// SIMATIC S7-200 project (STEP 7-Micro/WIN), CPU 226 CN REL 02.01

SYMBOL_TABLE 设备点名
烟气温度报警延时         T200
烟气温度报警限值         VD648
烟气压力保持数值         VD640
烟气流量保持数值         VD644
烟气温度保持数值         VD636
测量持续时间           T42
中间点3             V5010.2
中间点2             V5010.1
定时反吹持续时间         T39
后吹扫持续时间          T41
中间点1             V5010.0
干基折算粉尘浓度         VD632
测量               V1015.7
工况下烟气流量          VD608
烟气流速             VD616
Analyzer_Cali_FTE V6000.5
定时反吹_FTE         V6000.4
测量_FTE           V6000.3
后吹扫_FTE          V6000.2
采集背景_FTE         V6000.1
前吹扫_FTE          V6000.0
当前动作字符串输出        VB6100
Analyzer_Cali_STATU V1016.3
烟气温度低报警_STATU    V1012.6
维护切换_M           M1.0
手动_自动_M          M1.1
系统待机_M           M1.2
停止蜂鸣器_M          M1.3
手动启动             M1.4
探头反吹_M           M2.0
探头通零气_M          M2.1
探头通标气_M          M2.2
分析仪反吹_M          M2.3
分析仪通零气_M         M2.4
分析仪通标气_M         M2.5
手动采集背景_M         M2.6
测量_M             M2.7
蜂鸣器停止间隔时间        T40
报警指示灯_img        V1000.0
维护指示灯_img        V1000.1
运行指示灯_img        V1000.2
蜂鸣器_img          V1000.3
DCS报警信号_img      V1000.4
DCS运行信号_img      V1000.5
DCS维护信号_img      V1000.6
DCS待机信号_img      V1000.7
HOFI反吹电磁阀_img    V1001.0
三通电磁阀_img        V1001.1
氮气电磁阀_img        V1001.2
标气电磁阀_img        V1001.3
常开两通电磁阀_img      V1001.4
报警消除信号_img       V1004.0
DCS控制待机信号        V1004.2
探头反吹_ACT         V1006.0
探头通零气_ACT        V1006.1
探头通标气_ACT        V1006.2
分析仪反吹_ACT        V1006.3
分析仪通零气_ACT       V1006.4
分析仪通标气_ACT       V1006.5
采集背景_ACT         V1006.6
分析仪测量_ACT        V1006.7
探头后吹扫_ACT        V1007.0
分析仪前吹扫_ACT       V1007.1
定时反吹_ACT         V1007.2
Analyzer_Calibartion V1007.3
手动_自动_ACT        V1008.0
停止蜂鸣器_ACT        V1008.1
维护切换_ACT         V1008.4
待机_运行_ACT        V1008.5
启动报警_ACT         V1008.6
系统待机_ACT         V1008.7
系统运行_STATU       V1009.3
系统维护_STATU       V1009.4
系统报警_STATU       V1009.5
系统待机_STATU       V1009.6
手动_自动_STATU      V1010.6
蜂鸣器停止_运行_STATU   V1010.7
HOFI压力报警_STATU   V1011.0
HOFI温度报警_STATU   V1011.1
MDS压力报警_STATU    V1011.2
N2压力报警_STATU     V1011.3
粉尘仪报警_STATU      V1011.4
气路模块温度报警_STATU   V1011.5
加热管线温度报警_STATU   V1011.6
检测室温度报警_STATU    V1011.7
Reference失败报警_STATU V1012.0
检测室压力报警_STATU    V1012.1
文丘里压力报警_STATU    V1012.2
分析仪参数报警_STATU    V1012.3
分析仪报警_STATU      V1012.4
采样系统报警_STATU     V1012.5
联机通讯状警_STATU     V1012.7
采集背景_STATU       V1015.6
后吹扫_STATU        V1016.0
前吹扫_STATU        V1016.1
定时反吹_STATU       V1016.2
蜂鸣器启动中间变量        V5002.0
HCL折算            VD524
SO2折算            VD528
NOx折算            VD532
NH3折算            VD536
NO折算             VD540
NO2折算            VD544
SO2实测值           VD548
HF折算             VD552
CO折算             VD556
CO2折算            VD560
NOX实测值           VD564
水分含量             VD568
湿氧浓度             VD576
检测室压力            VD580
文丘里压力            VD584
烟气温度             VD592
烟气压力             VD596
烟气压差             VD600
粉尘浓度             VD604
干基标准烟气流量         VD620
标态粉尘浓度           VD624
干氧浓度             VD628
检测室压力_img        VW900
文丘里压力_img        VW902
湿氧浓度_img         VW904
烟气温度_img         VW906
烟气压差_img         VW908
烟气压力_img         VW910
粉尘浓度_img         VW912
END_SYMBOL_TABLE

ORGANIZATION_BLOCK Main:OB1
TITLE=
// //增加氧气修正及烟气流量，粉尘修正的计算
// //模拟量输出量程设置
// //增加定时反吹定时时间 配合组态用于MBGAS3000驱动
// //Define Action子程序，增加报警状态点 V1009.5  网络16,17
// //Define Action子程序，修改1008.5为待机_运行控制点，输出状态为系统待机， 网络14,15
// //Operation & Remove Operation子程序增加V1000.7信号的置位与复位
// 
// //修改干基计算子模块为标态计算
// 
// //采样系统报警时也可执行待机动作
// 
// //增加profibusDP数据通信功能
// 
// 
BEGIN
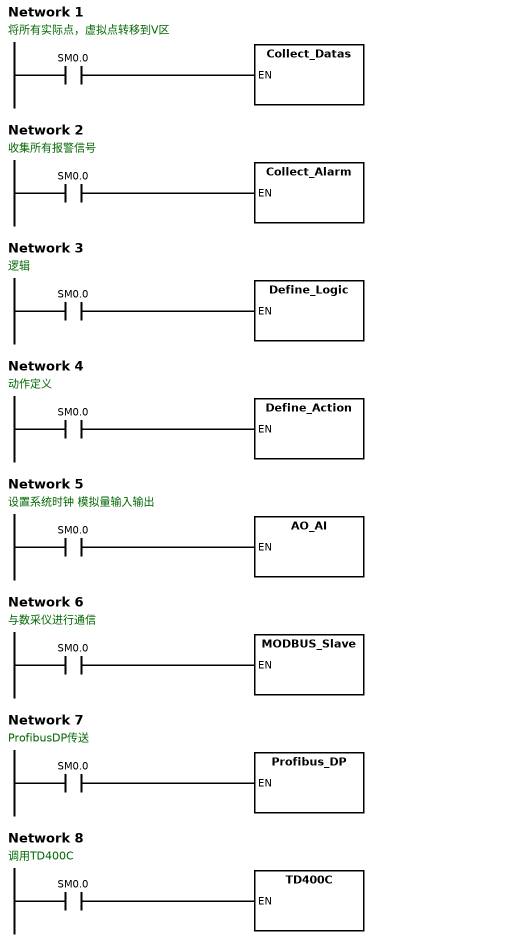
Network 1
// 将所有实际点，虚拟点转移到V区
LD     SM0.0
CALL   Collect_Datas:SBR7
Network 2
// 收集所有报警信号
LD     SM0.0
CALL   Collect_Alarm:SBR8
Network 3
// 逻辑
LD     SM0.0
CALL   Define_Logic:SBR10
Network 4
// 动作定义
LD     SM0.0
CALL   Define_Action:SBR9
Network 5
// 设置系统时钟 模拟量输入输出
LD     SM0.0
CALL   AO_AI:SBR15
Network 6
// 与数采仪进行通信
LD     SM0.0
CALL   MODBUS_Slave:SBR21
Network 7
// ProfibusDP传送
LD     SM0.0
CALL   Profibus_DP:SBR25
Network 8
// 调用TD400C
LD     SM0.0
CALL   TD400C:SBR16
END_ORGANIZATION_BLOCK

// SBR0: protected block, not included

SUBROUTINE_BLOCK Alarm:SBR1
TITLE=报警执行动作
BEGIN
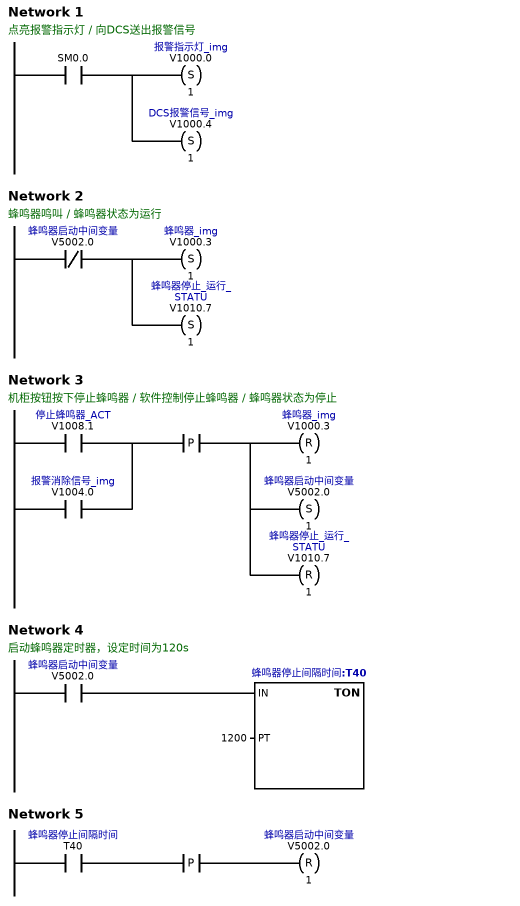
Network 1
// 点亮报警指示灯
// 向DCS送出报警信号
LD     SM0.0
S      报警指示灯_img:V1000.0, 1
S      DCS报警信号_img:V1000.4, 1
Network 2
// 蜂鸣器鸣叫
// 蜂鸣器状态为运行
LDN    蜂鸣器启动中间变量:V5002.0
S      蜂鸣器_img:V1000.3, 1
S      蜂鸣器停止_运行_STATU:V1010.7, 1
Network 3
// 机柜按钮按下停止蜂鸣器
// 软件控制停止蜂鸣器
// 蜂鸣器状态为停止
LD     停止蜂鸣器_ACT:V1008.1
O      报警消除信号_img:V1004.0
EU
R      蜂鸣器_img:V1000.3, 1
S      蜂鸣器启动中间变量:V5002.0, 1
R      蜂鸣器停止_运行_STATU:V1010.7, 1
Network 4
// 启动蜂鸣器定时器，设定时间为120s
LD     蜂鸣器启动中间变量:V5002.0
TON    蜂鸣器停止间隔时间:T40, 1200
Network 5
LD     蜂鸣器停止间隔时间:T40
EU
R      蜂鸣器启动中间变量:V5002.0, 1
END_SUBROUTINE_BLOCK

SUBROUTINE_BLOCK Remove_Alarm:SBR2
TITLE=报警消除后执行动作
BEGIN
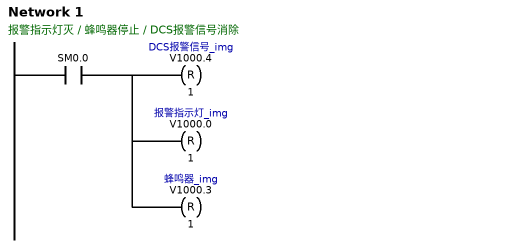
Network 1
// 报警指示灯灭
// 蜂鸣器停止
// DCS报警信号消除
LD     SM0.0
R      DCS报警信号_img:V1000.4, 1
R      报警指示灯_img:V1000.0, 1
R      蜂鸣器_img:V1000.3, 1
END_SUBROUTINE_BLOCK

SUBROUTINE_BLOCK Operation:SBR3
TITLE=子程序注释
BEGIN
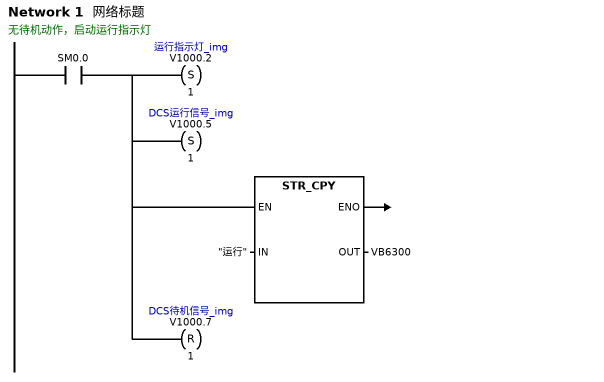
Network 1 // 网络标题
// 无待机动作，启动运行指示灯
LD     SM0.0
S      运行指示灯_img:V1000.2, 1
S      DCS运行信号_img:V1000.5, 1
SCPY   "运行", VB6300
R      DCS待机信号_img:V1000.7, 1
END_SUBROUTINE_BLOCK

SUBROUTINE_BLOCK Remove_Operation:SBR4
TITLE=子程序注释
BEGIN
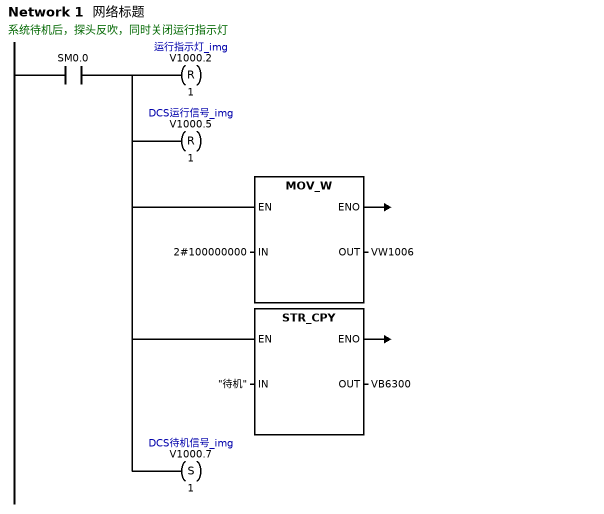
Network 1 // 网络标题
// 系统待机后，探头反吹，同时关闭运行指示灯
LD     SM0.0
R      运行指示灯_img:V1000.2, 1
R      DCS运行信号_img:V1000.5, 1
MOVW   2#100000000, VW1006
SCPY   "待机", VB6300
S      DCS待机信号_img:V1000.7, 1
Network 11 // 网络标题
// 网络注释
END_SUBROUTINE_BLOCK

SUBROUTINE_BLOCK Maintenance:SBR5
TITLE=子程序注释
BEGIN
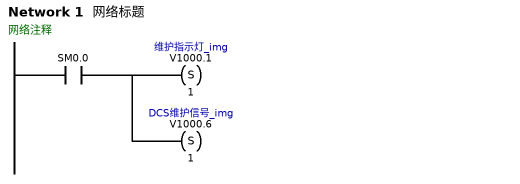
Network 1 // 网络标题
// 网络注释
LD     SM0.0
S      维护指示灯_img:V1000.1, 1
S      DCS维护信号_img:V1000.6, 1
END_SUBROUTINE_BLOCK

SUBROUTINE_BLOCK Remove_Maintenance:SBR6
TITLE=子程序注释
BEGIN
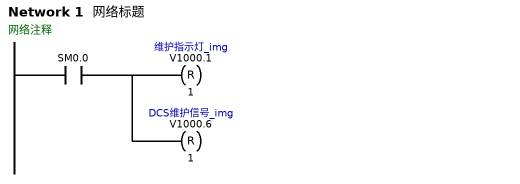
Network 1 // 网络标题
// 网络注释
LD     SM0.0
R      维护指示灯_img:V1000.1, 1
R      DCS维护信号_img:V1000.6, 1
END_SUBROUTINE_BLOCK

SUBROUTINE_BLOCK Collect_Datas:SBR7
TITLE=数据转移V区
BEGIN
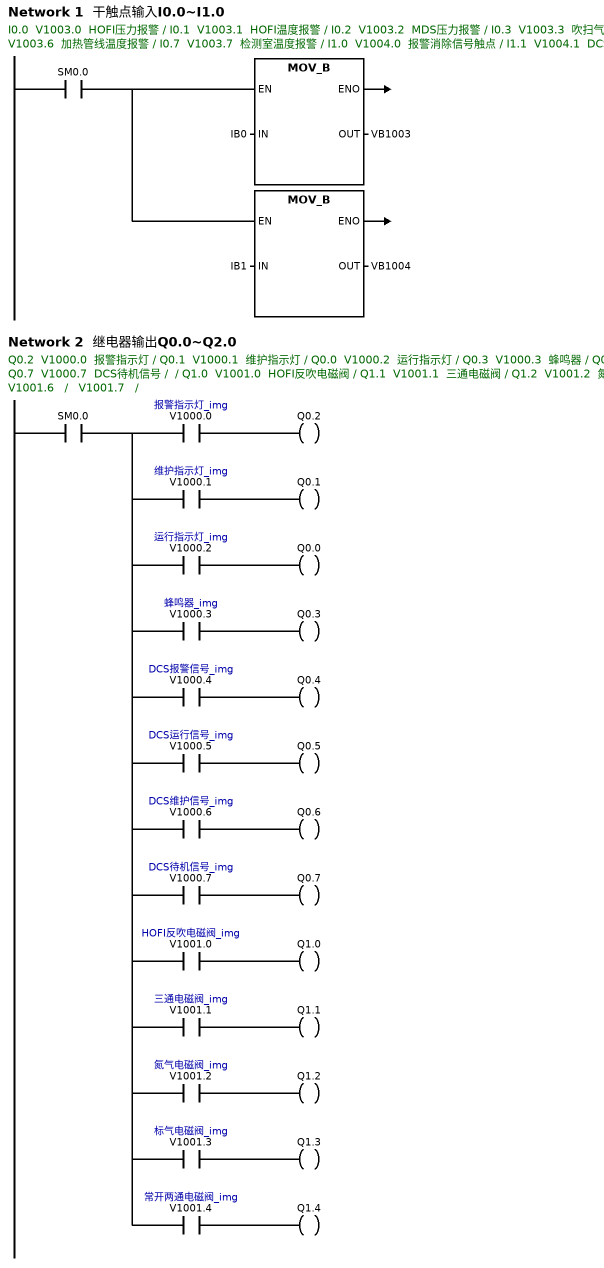
Network 1 // 干触点输入I0.0~I1.0
// I0.0	V1003.0	HOFI压力报警
// I0.1	V1003.1	HOFI温度报警
// I0.2	V1003.2	MDS压力报警
// I0.3	V1003.3	吹扫气体发生器输出压力报警
// I0.4	V1003.4	粉尘仪报警
// I0.5	V1003.5	分析仪采样模块温度报警
// I0.6	V1003.6	加热管线温度报警
// I0.7	V1003.7	检测室温度报警
// I1.0	V1004.0	报警消除信号触点
// I1.1	V1004.1	DCS控制系统采样信号
// I1.2	V1004.2	DCS控制系统待机信号
LD     SM0.0
MOVB   IB0, VB1003
MOVB   IB1, VB1004
Network 2 // 继电器输出Q0.0~Q2.0
// Q0.2	V1000.0	报警指示灯
// Q0.1	V1000.1	维护指示灯
// Q0.0	V1000.2	运行指示灯
// Q0.3	V1000.3	蜂鸣器
// Q0.4	V1000.4	DCS报警信号
// Q0.5	V1000.5	DCS运行信号
// Q0.6	V1000.6	DCS维护信号
// Q0.7	V1000.7	DCS待机信号
// 
// Q1.0	V1001.0	HOFI反吹电磁阀
// Q1.1	V1001.1	三通电磁阀
// Q1.2	V1001.2	氮气电磁阀
// Q1.3	V1001.3	标气电磁阀
// Q1.4	V1001.4	常开两通电磁阀
// 	V1001.5	
// 	V1001.6	
// 	V1001.7	
// 
LD     SM0.0
LPS
A      报警指示灯_img:V1000.0
=      Q0.2
LRD
A      维护指示灯_img:V1000.1
=      Q0.1
LRD
A      运行指示灯_img:V1000.2
=      Q0.0
LRD
A      蜂鸣器_img:V1000.3
=      Q0.3
LRD
A      DCS报警信号_img:V1000.4
=      Q0.4
LRD
A      DCS运行信号_img:V1000.5
=      Q0.5
LRD
A      DCS维护信号_img:V1000.6
=      Q0.6
LRD
A      DCS待机信号_img:V1000.7
=      Q0.7
LRD
A      HOFI反吹电磁阀_img:V1001.0
=      Q1.0
LRD
A      三通电磁阀_img:V1001.1
=      Q1.1
LRD
A      氮气电磁阀_img:V1001.2
=      Q1.2
LRD
A      标气电磁阀_img:V1001.3
=      Q1.3
LPP
A      常开两通电磁阀_img:V1001.4
=      Q1.4
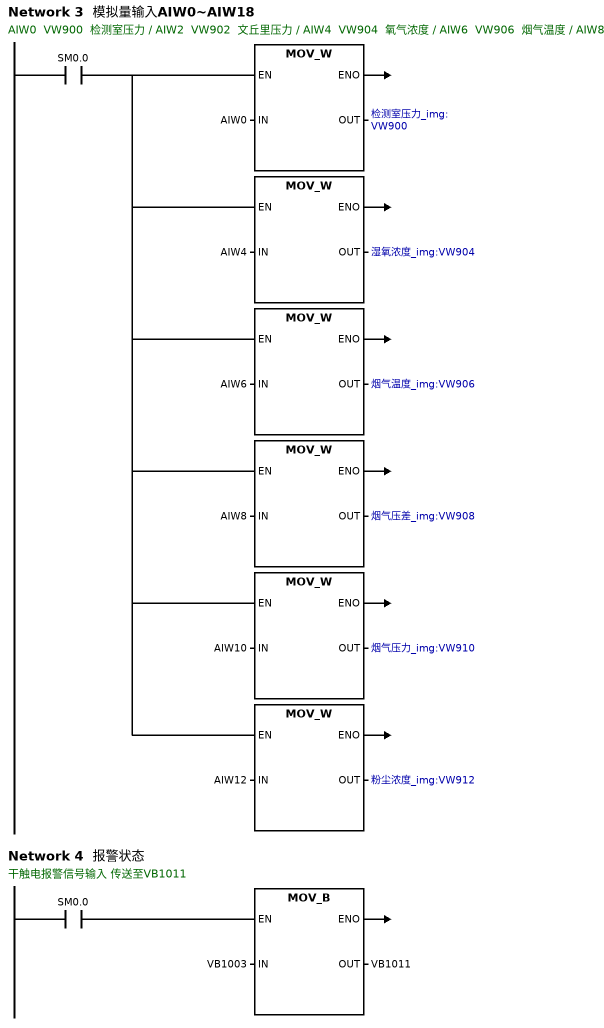
Network 3 // 模拟量输入AIW0~AIW18
// AIW0	VW900	检测室压力
// AIW2	VW902	文丘里压力
// AIW4	VW904	氧气浓度
// AIW6	VW906	烟气温度
// AIW8	VW908	烟气压差
// AIW10	VW910	烟气压力
// AIW12	VW912	粉尘浓度/不透光度
// 
LD     SM0.0
MOVW   AIW0, 检测室压力_img:VW900
MOVW   AIW4, 湿氧浓度_img:VW904
MOVW   AIW6, 烟气温度_img:VW906
MOVW   AIW8, 烟气压差_img:VW908
MOVW   AIW10, 烟气压力_img:VW910
MOVW   AIW12, 粉尘浓度_img:VW912
Network 4 // 报警状态
// 干触电报警信号输入 传送至VB1011
LD     SM0.0
MOVB   VB1003, VB1011
END_SUBROUTINE_BLOCK

SUBROUTINE_BLOCK Collect_Alarm:SBR8
TITLE=
BEGIN
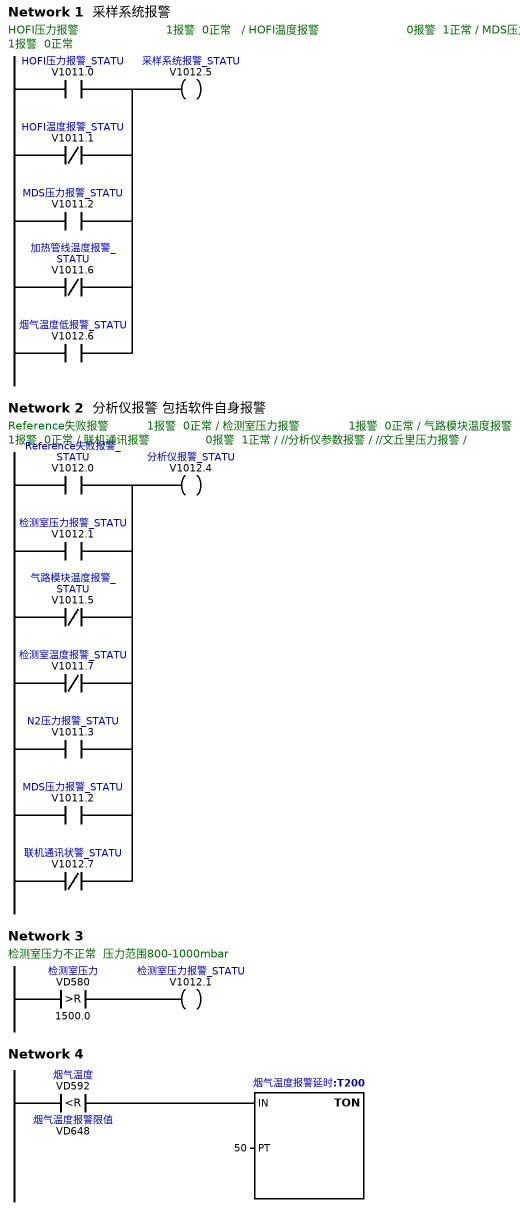
Network 1 // 采样系统报警
// HOFI压力报警                         1报警  0正常  
// HOFI温度报警                         0报警  1正常
// MDS压力报警                          1报警  0正常
// 加热管线温度报警                     0报警  1正常
// 烟气温度低                           1报警  0正常
LD     HOFI压力报警_STATU:V1011.0
ON     HOFI温度报警_STATU:V1011.1
O      MDS压力报警_STATU:V1011.2
ON     加热管线温度报警_STATU:V1011.6
O      烟气温度低报警_STATU:V1012.6
=      采样系统报警_STATU:V1012.5
Network 2 // 分析仪报警 包括软件自身报警
// Reference失败报警           1报警  0正常
// 检测室压力报警              1报警  0正常
// 气路模块温度报警            0报警  1正常
// 检测室温度报警              0报警  1正常
// N2压力报警                  1报警  0正常
// MDS压力报警                 1报警  0正常
// 联机通讯报警                0报警  1正常
// //分析仪参数报警
// //文丘里压力报警
// 
LD     Reference失败报警_STATU:V1012.0
O      检测室压力报警_STATU:V1012.1
ON     气路模块温度报警_STATU:V1011.5
ON     检测室温度报警_STATU:V1011.7
O      N2压力报警_STATU:V1011.3
O      MDS压力报警_STATU:V1011.2
ON     联机通讯状警_STATU:V1012.7
=      分析仪报警_STATU:V1012.4
Network 3
// 检测室压力不正常  压力范围800-1000mbar
LDR>   检测室压力:VD580, 1500.0
=      检测室压力报警_STATU:V1012.1
Network 4
LDR<   烟气温度:VD592, 烟气温度报警限值:VD648
TON    烟气温度报警延时:T200, 50
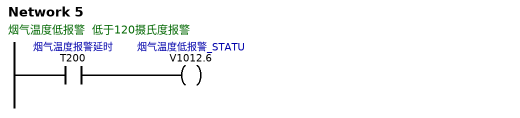
Network 5
// 烟气温度低报警  低于120摄氏度报警
LD     烟气温度报警延时:T200
=      烟气温度低报警_STATU:V1012.6
END_SUBROUTINE_BLOCK

SUBROUTINE_BLOCK Define_Action:SBR9
TITLE=
BEGIN
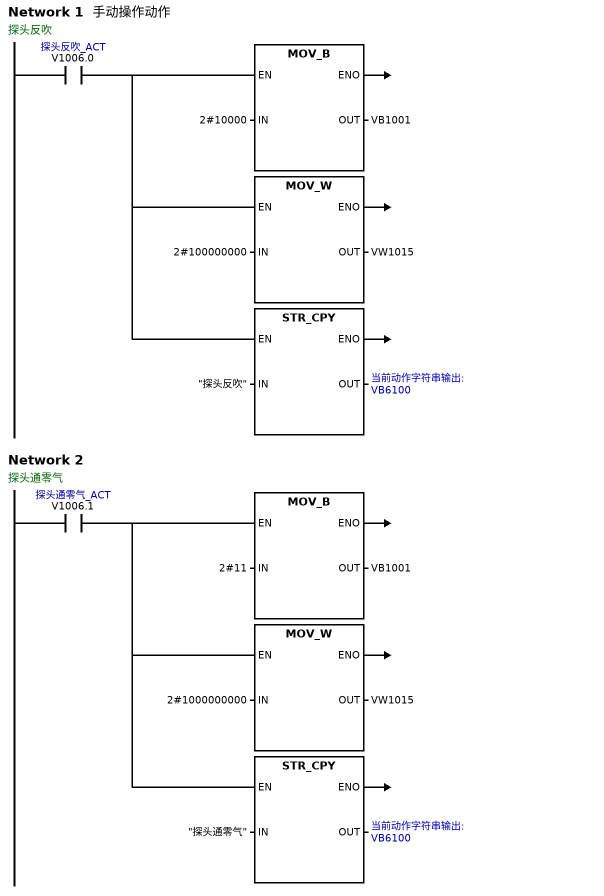
Network 1 // 手动操作动作
// 探头反吹
LD     探头反吹_ACT:V1006.0
MOVB   2#10000, VB1001
MOVW   2#100000000, VW1015
SCPY   "探头反吹", 当前动作字符串输出:VB6100
Network 2
// 探头通零气
LD     探头通零气_ACT:V1006.1
MOVB   2#11, VB1001
MOVW   2#1000000000, VW1015
SCPY   "探头通零气", 当前动作字符串输出:VB6100
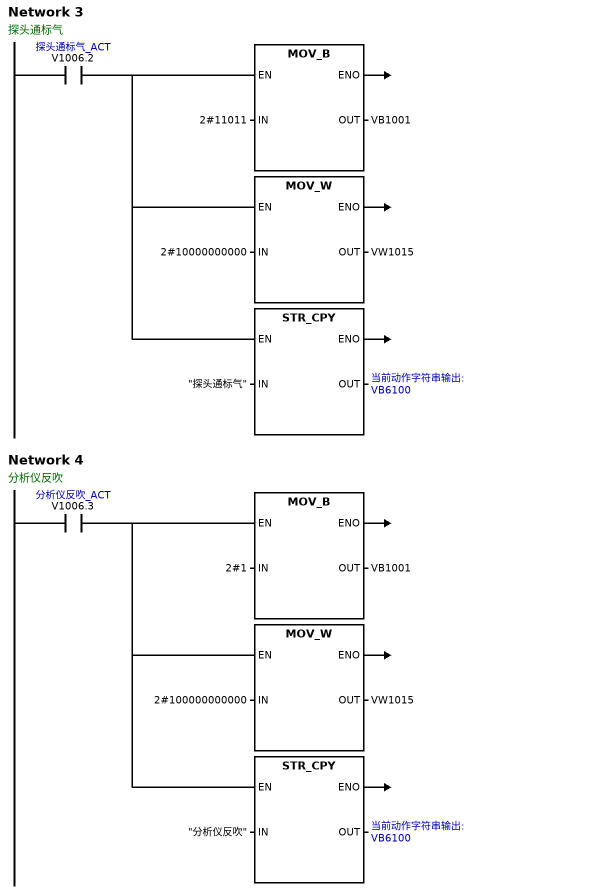
Network 3
// 探头通标气
LD     探头通标气_ACT:V1006.2
MOVB   2#11011, VB1001
MOVW   2#10000000000, VW1015
SCPY   "探头通标气", 当前动作字符串输出:VB6100
Network 4
// 分析仪反吹
LD     分析仪反吹_ACT:V1006.3
MOVB   2#1, VB1001
MOVW   2#100000000000, VW1015
SCPY   "分析仪反吹", 当前动作字符串输出:VB6100
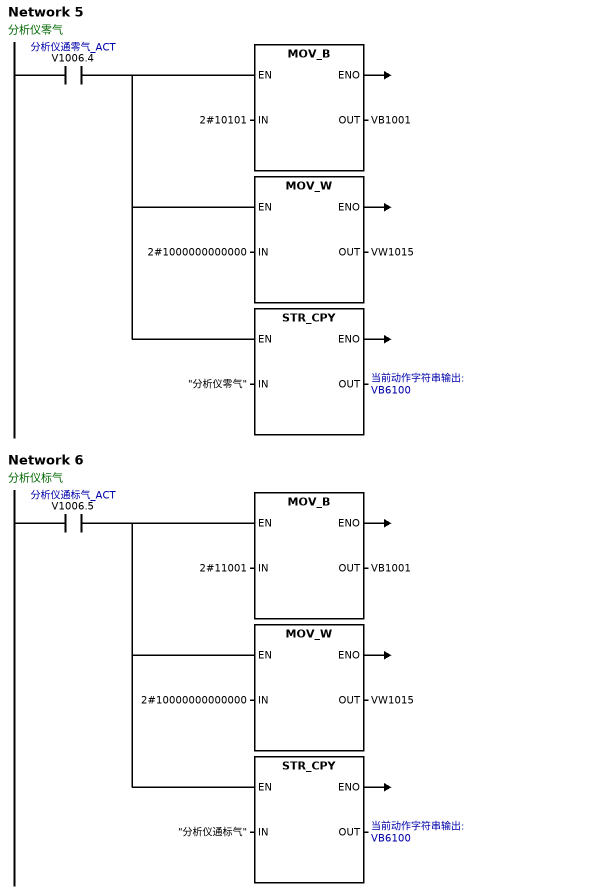
Network 5
// 分析仪零气
LD     分析仪通零气_ACT:V1006.4
MOVB   2#10101, VB1001
MOVW   2#1000000000000, VW1015
SCPY   "分析仪零气", 当前动作字符串输出:VB6100
Network 6
// 分析仪标气
LD     分析仪通标气_ACT:V1006.5
MOVB   2#11001, VB1001
MOVW   2#10000000000000, VW1015
SCPY   "分析仪通标气", 当前动作字符串输出:VB6100
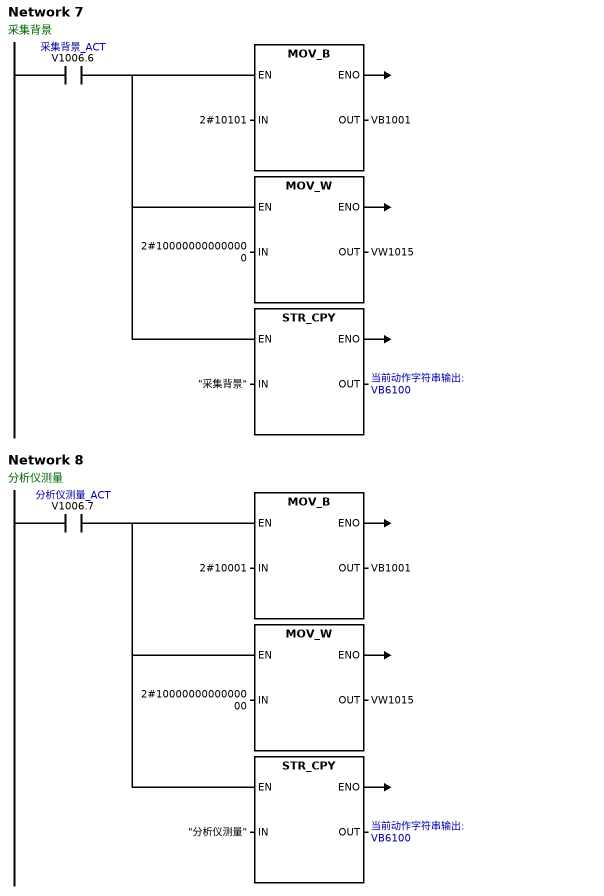
Network 7
// 采集背景
LD     采集背景_ACT:V1006.6
MOVB   2#10101, VB1001
MOVW   2#100000000000000, VW1015
SCPY   "采集背景", 当前动作字符串输出:VB6100
Network 8
// 分析仪测量
LD     分析仪测量_ACT:V1006.7
MOVB   2#10001, VB1001
MOVW   2#1000000000000000, VW1015
SCPY   "分析仪测量", 当前动作字符串输出:VB6100
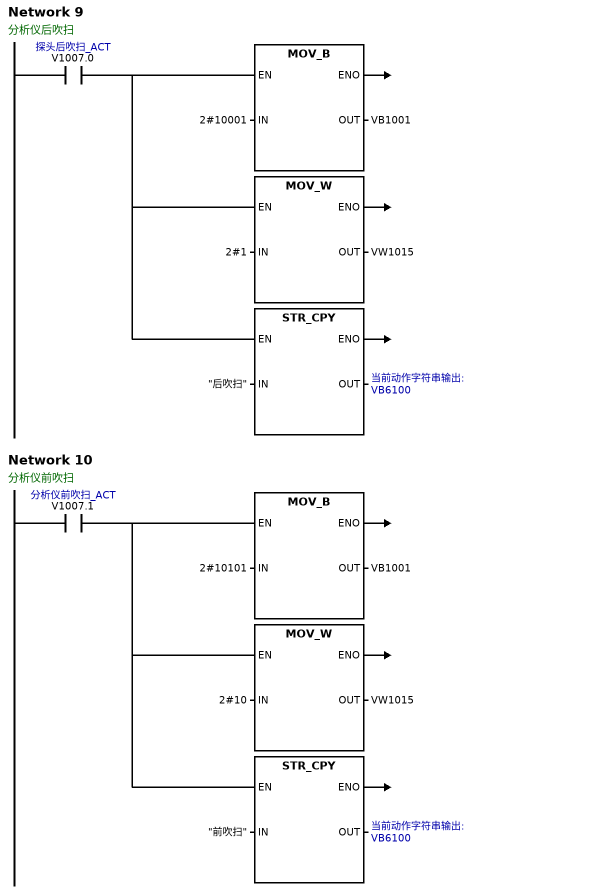
Network 9
// 分析仪后吹扫
LD     探头后吹扫_ACT:V1007.0
MOVB   2#10001, VB1001
MOVW   2#1, VW1015
SCPY   "后吹扫", 当前动作字符串输出:VB6100
Network 10
// 分析仪前吹扫
LD     分析仪前吹扫_ACT:V1007.1
MOVB   2#10101, VB1001
MOVW   2#10, VW1015
SCPY   "前吹扫", 当前动作字符串输出:VB6100
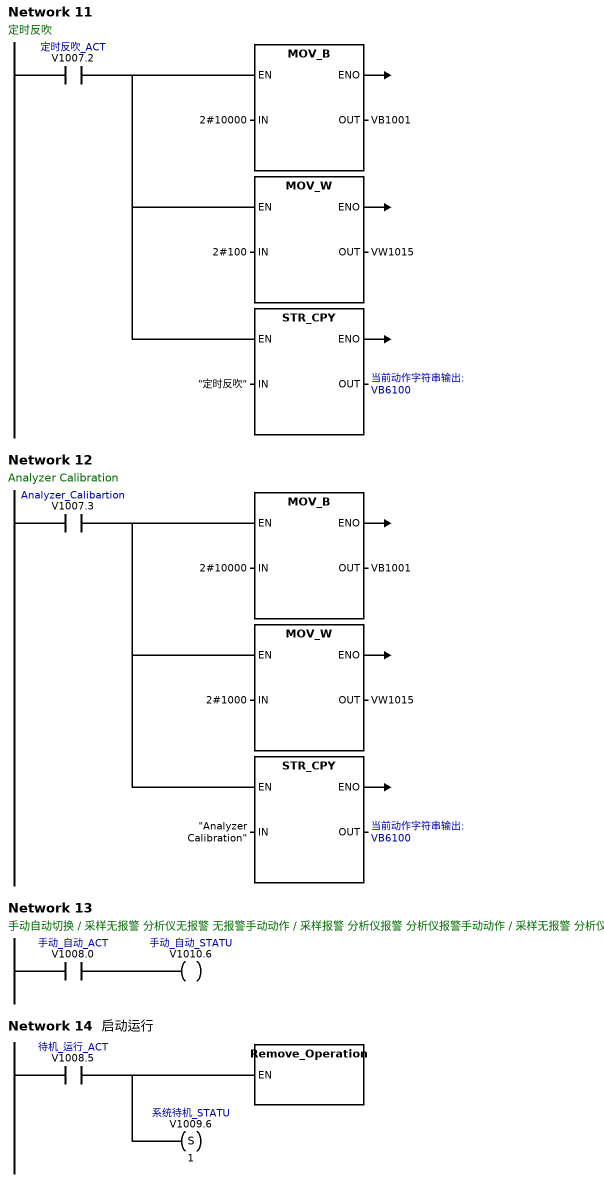
Network 11
// 定时反吹
LD     定时反吹_ACT:V1007.2
MOVB   2#10000, VB1001
MOVW   2#100, VW1015
SCPY   "定时反吹", 当前动作字符串输出:VB6100
Network 12
// Analyzer Calibration
LD     Analyzer_Calibartion:V1007.3
MOVB   2#10000, VB1001
MOVW   2#1000, VW1015
SCPY   "Analyzer Calibration", 当前动作字符串输出:VB6100
Network 13
// 手动自动切换
// 采样无报警 分析仪无报警 无报警手动动作
// 采样报警 分析仪报警 分析仪报警手动动作
// 采样无报警 分析仪报警 分析仪报警手动动作
// 采样报警 分析仪无报警 探头报警手动动作
LD     手动_自动_ACT:V1008.0
=      手动_自动_STATU:V1010.6
Network 14 // 启动运行
LD     待机_运行_ACT:V1008.5
CALL   Remove_Operation:SBR4
S      系统待机_STATU:V1009.6, 1
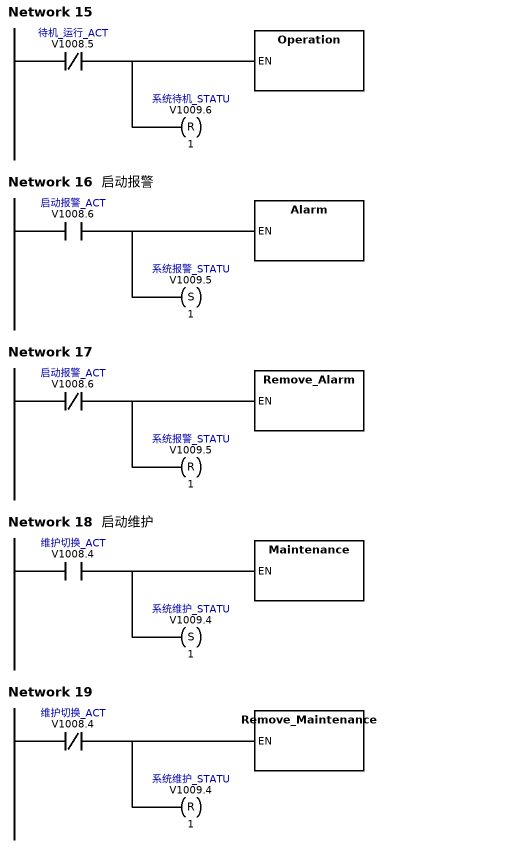
Network 15
LDN    待机_运行_ACT:V1008.5
CALL   Operation:SBR3
R      系统待机_STATU:V1009.6, 1
Network 16 // 启动报警
LD     启动报警_ACT:V1008.6
CALL   Alarm:SBR1
S      系统报警_STATU:V1009.5, 1
Network 17
LDN    启动报警_ACT:V1008.6
CALL   Remove_Alarm:SBR2
R      系统报警_STATU:V1009.5, 1
Network 18 // 启动维护
LD     维护切换_ACT:V1008.4
CALL   Maintenance:SBR5
S      系统维护_STATU:V1009.4, 1
Network 19
LDN    维护切换_ACT:V1008.4
CALL   Remove_Maintenance:SBR6
R      系统维护_STATU:V1009.4, 1
END_SUBROUTINE_BLOCK

SUBROUTINE_BLOCK Define_Logic:SBR10
TITLE=
BEGIN
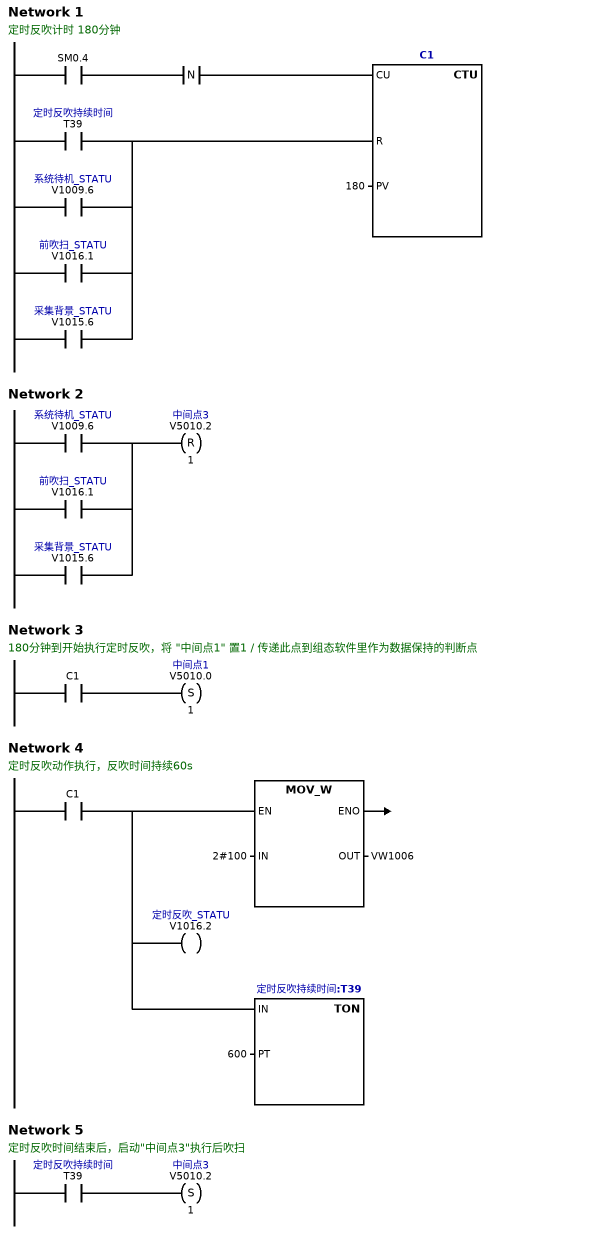
Network 1
// 定时反吹计时 180分钟
LD     SM0.4
ED
LD     定时反吹持续时间:T39
O      系统待机_STATU:V1009.6
O      前吹扫_STATU:V1016.1
O      采集背景_STATU:V1015.6
CTU    C1, 180
Network 2
LD     系统待机_STATU:V1009.6
O      前吹扫_STATU:V1016.1
O      采集背景_STATU:V1015.6
R      中间点3:V5010.2, 1
Network 3
// 180分钟到开始执行定时反吹，将 "中间点1" 置1
// 传递此点到组态软件里作为数据保持的判断点
LD     C1
S      中间点1:V5010.0, 1
Network 4
// 定时反吹动作执行，反吹时间持续60s
LD     C1
MOVW   2#100, VW1006
=      定时反吹_STATU:V1016.2
TON    定时反吹持续时间:T39, 600
Network 5
// 定时反吹时间结束后，启动"中间点3"执行后吹扫
LD     定时反吹持续时间:T39
S      中间点3:V5010.2, 1
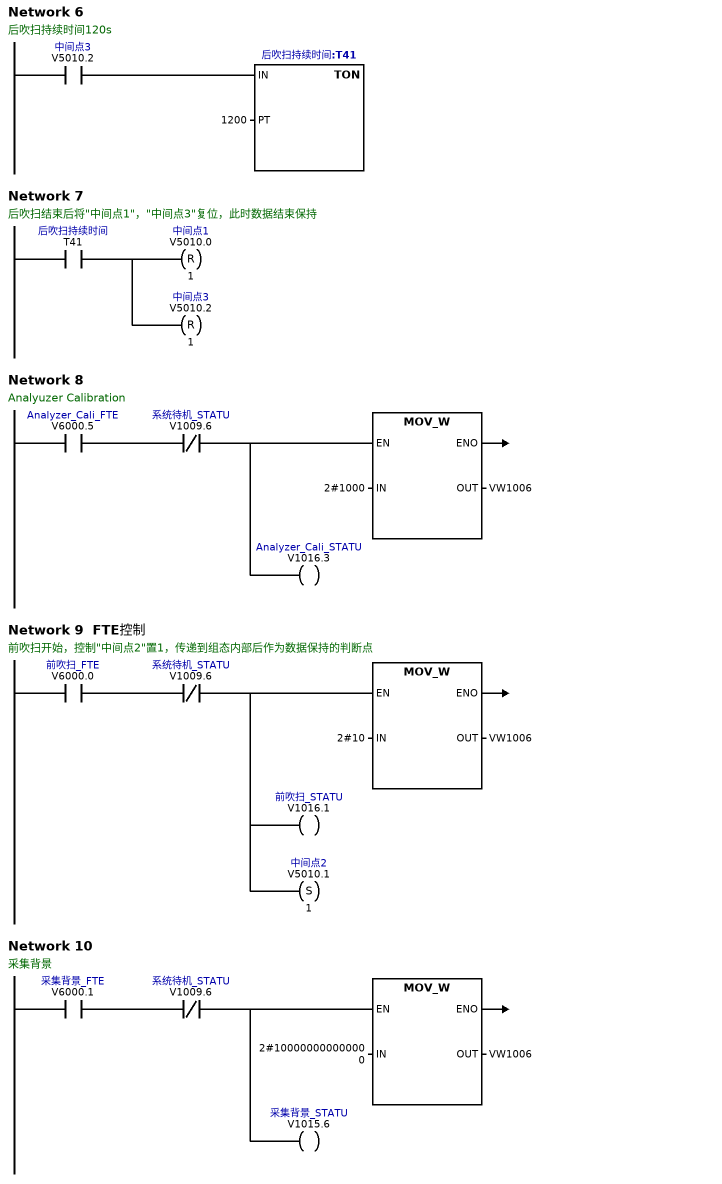
Network 6
// 后吹扫持续时间120s
LD     中间点3:V5010.2
TON    后吹扫持续时间:T41, 1200
Network 7
// 后吹扫结束后将"中间点1"，"中间点3"复位，此时数据结束保持
LD     后吹扫持续时间:T41
R      中间点1:V5010.0, 1
R      中间点3:V5010.2, 1
Network 8
// Analyuzer Calibration
LD     Analyzer_Cali_FTE:V6000.5
AN     系统待机_STATU:V1009.6
MOVW   2#1000, VW1006
=      Analyzer_Cali_STATU:V1016.3
Network 9 // FTE控制
// 前吹扫开始，控制"中间点2"置1，传递到组态内部后作为数据保持的判断点
LD     前吹扫_FTE:V6000.0
AN     系统待机_STATU:V1009.6
MOVW   2#10, VW1006
=      前吹扫_STATU:V1016.1
S      中间点2:V5010.1, 1
Network 10
// 采集背景
LD     采集背景_FTE:V6000.1
AN     系统待机_STATU:V1009.6
MOVW   2#100000000000000, VW1006
=      采集背景_STATU:V1015.6
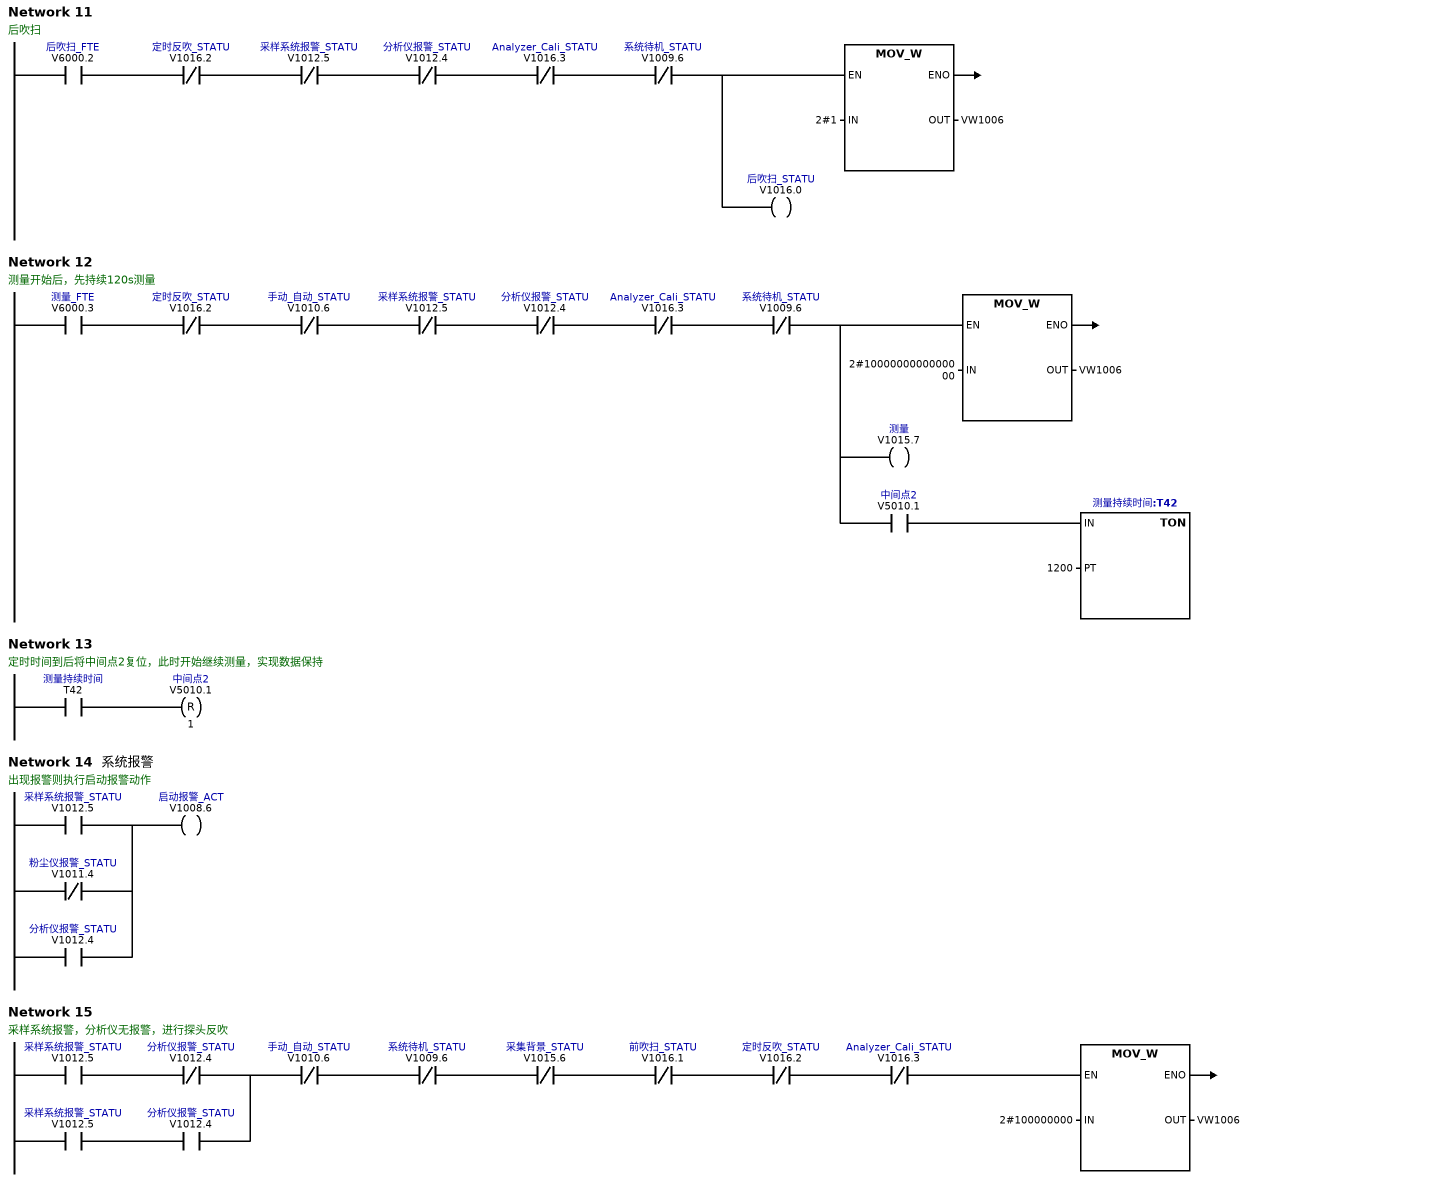
Network 11
// 后吹扫
LD     后吹扫_FTE:V6000.2
AN     定时反吹_STATU:V1016.2
AN     采样系统报警_STATU:V1012.5
AN     分析仪报警_STATU:V1012.4
AN     Analyzer_Cali_STATU:V1016.3
AN     系统待机_STATU:V1009.6
MOVW   2#1, VW1006
=      后吹扫_STATU:V1016.0
Network 12
// 测量开始后，先持续120s测量
LD     测量_FTE:V6000.3
AN     定时反吹_STATU:V1016.2
AN     手动_自动_STATU:V1010.6
AN     采样系统报警_STATU:V1012.5
AN     分析仪报警_STATU:V1012.4
AN     Analyzer_Cali_STATU:V1016.3
AN     系统待机_STATU:V1009.6
MOVW   2#1000000000000000, VW1006
=      测量:V1015.7
A      中间点2:V5010.1
TON    测量持续时间:T42, 1200
Network 13
// 定时时间到后将中间点2复位，此时开始继续测量，实现数据保持
LD     测量持续时间:T42
R      中间点2:V5010.1, 1
Network 14 // 系统报警
// 出现报警则执行启动报警动作
LD     采样系统报警_STATU:V1012.5
ON     粉尘仪报警_STATU:V1011.4
O      分析仪报警_STATU:V1012.4
=      启动报警_ACT:V1008.6
Network 15
// 采样系统报警，分析仪无报警，进行探头反吹
LD     采样系统报警_STATU:V1012.5
AN     分析仪报警_STATU:V1012.4
LD     采样系统报警_STATU:V1012.5
A      分析仪报警_STATU:V1012.4
OLD
AN     手动_自动_STATU:V1010.6
AN     系统待机_STATU:V1009.6
AN     采集背景_STATU:V1015.6
AN     前吹扫_STATU:V1016.1
AN     定时反吹_STATU:V1016.2
AN     Analyzer_Cali_STATU:V1016.3
MOVW   2#100000000, VW1006
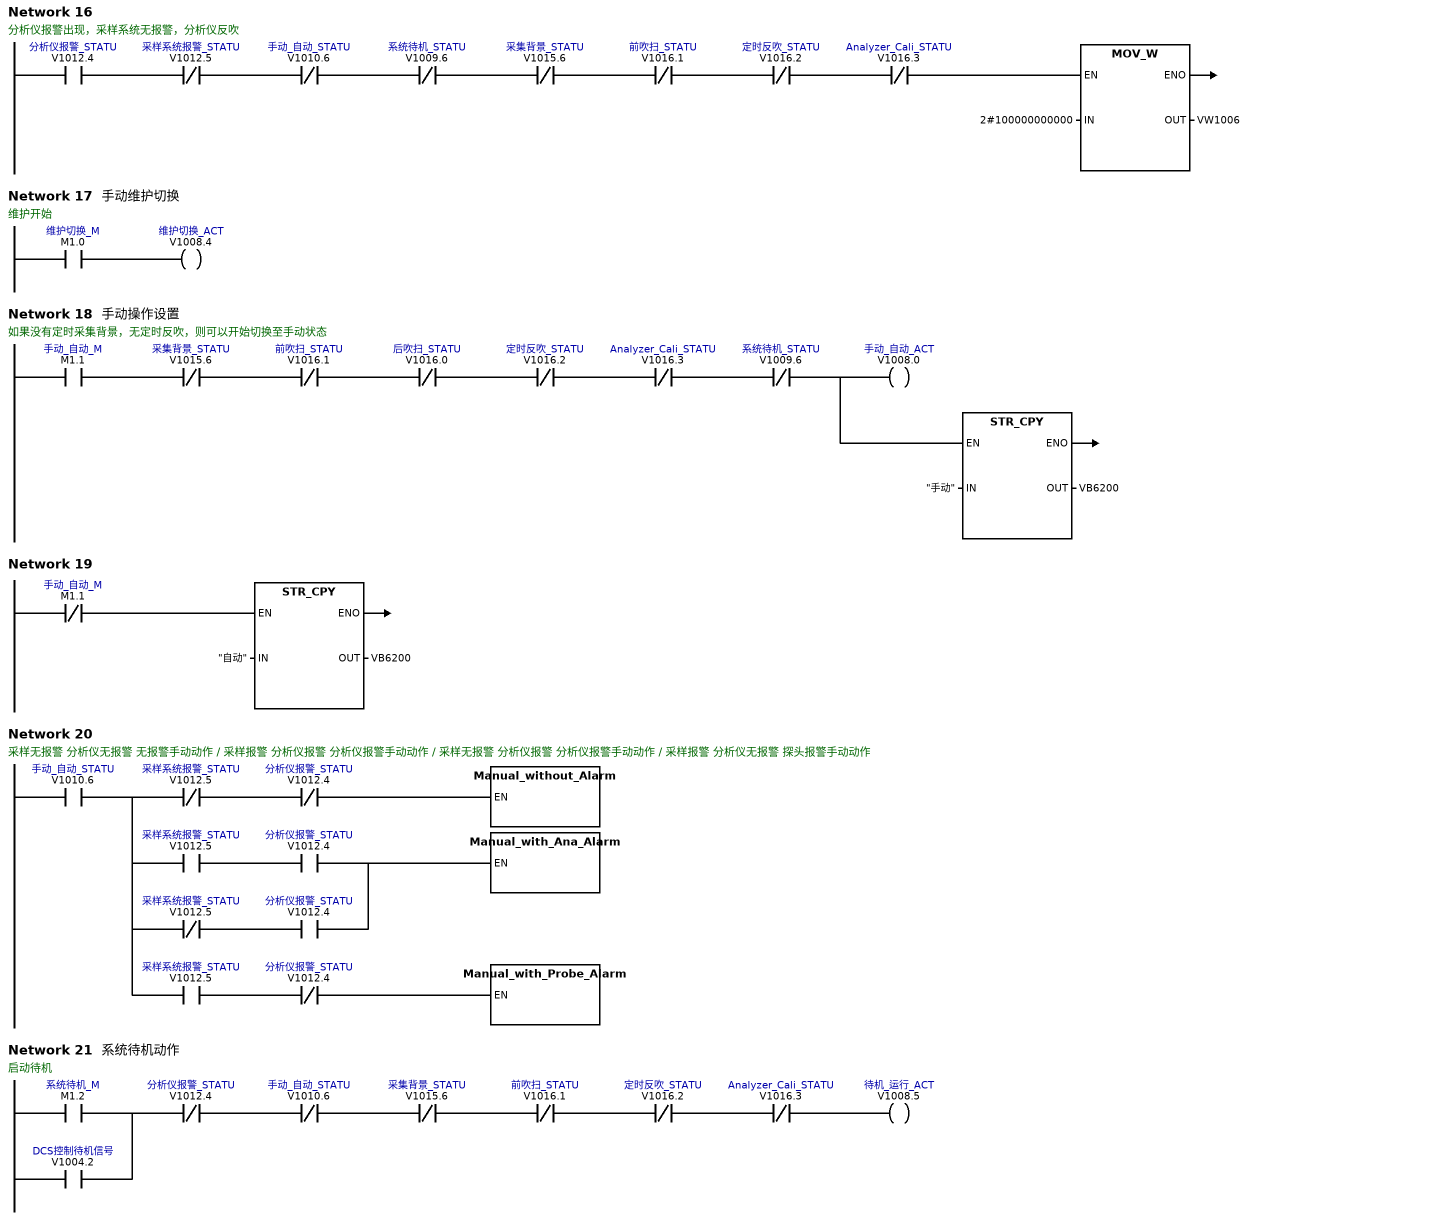
Network 16
// 分析仪报警出现，采样系统无报警，分析仪反吹
LD     分析仪报警_STATU:V1012.4
AN     采样系统报警_STATU:V1012.5
AN     手动_自动_STATU:V1010.6
AN     系统待机_STATU:V1009.6
AN     采集背景_STATU:V1015.6
AN     前吹扫_STATU:V1016.1
AN     定时反吹_STATU:V1016.2
AN     Analyzer_Cali_STATU:V1016.3
MOVW   2#100000000000, VW1006
Network 17 // 手动维护切换
// 维护开始
LD     维护切换_M:M1.0
=      维护切换_ACT:V1008.4
Network 18 // 手动操作设置
// 如果没有定时采集背景，无定时反吹，则可以开始切换至手动状态
LD     手动_自动_M:M1.1
AN     采集背景_STATU:V1015.6
AN     前吹扫_STATU:V1016.1
AN     后吹扫_STATU:V1016.0
AN     定时反吹_STATU:V1016.2
AN     Analyzer_Cali_STATU:V1016.3
AN     系统待机_STATU:V1009.6
=      手动_自动_ACT:V1008.0
SCPY   "手动", VB6200
Network 19
LDN    手动_自动_M:M1.1
SCPY   "自动", VB6200
Network 20
// 采样无报警 分析仪无报警 无报警手动动作
// 采样报警 分析仪报警 分析仪报警手动动作
// 采样无报警 分析仪报警 分析仪报警手动动作
// 采样报警 分析仪无报警 探头报警手动动作
LD     手动_自动_STATU:V1010.6
LPS
AN     采样系统报警_STATU:V1012.5
AN     分析仪报警_STATU:V1012.4
CALL   Manual_without_Alarm:SBR12
LRD
LD     采样系统报警_STATU:V1012.5
A      分析仪报警_STATU:V1012.4
LDN    采样系统报警_STATU:V1012.5
A      分析仪报警_STATU:V1012.4
OLD
ALD
CALL   Manual_with_Ana_Alarm:SBR13
LPP
A      采样系统报警_STATU:V1012.5
AN     分析仪报警_STATU:V1012.4
CALL   Manual_with_Probe_Alarm:SBR14
Network 21 // 系统待机动作
// 启动待机
LD     系统待机_M:M1.2
O      DCS控制待机信号:V1004.2
AN     分析仪报警_STATU:V1012.4
AN     手动_自动_STATU:V1010.6
AN     采集背景_STATU:V1015.6
AN     前吹扫_STATU:V1016.1
AN     定时反吹_STATU:V1016.2
AN     Analyzer_Cali_STATU:V1016.3
=      待机_运行_ACT:V1008.5
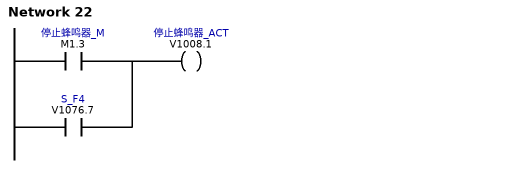
Network 22
LD     停止蜂鸣器_M:M1.3
O      S_F4:V1076.7
=      停止蜂鸣器_ACT:V1008.1
END_SUBROUTINE_BLOCK

// SBR11: protected block, not included

SUBROUTINE_BLOCK Manual_without_Alarm:SBR12
TITLE=
BEGIN
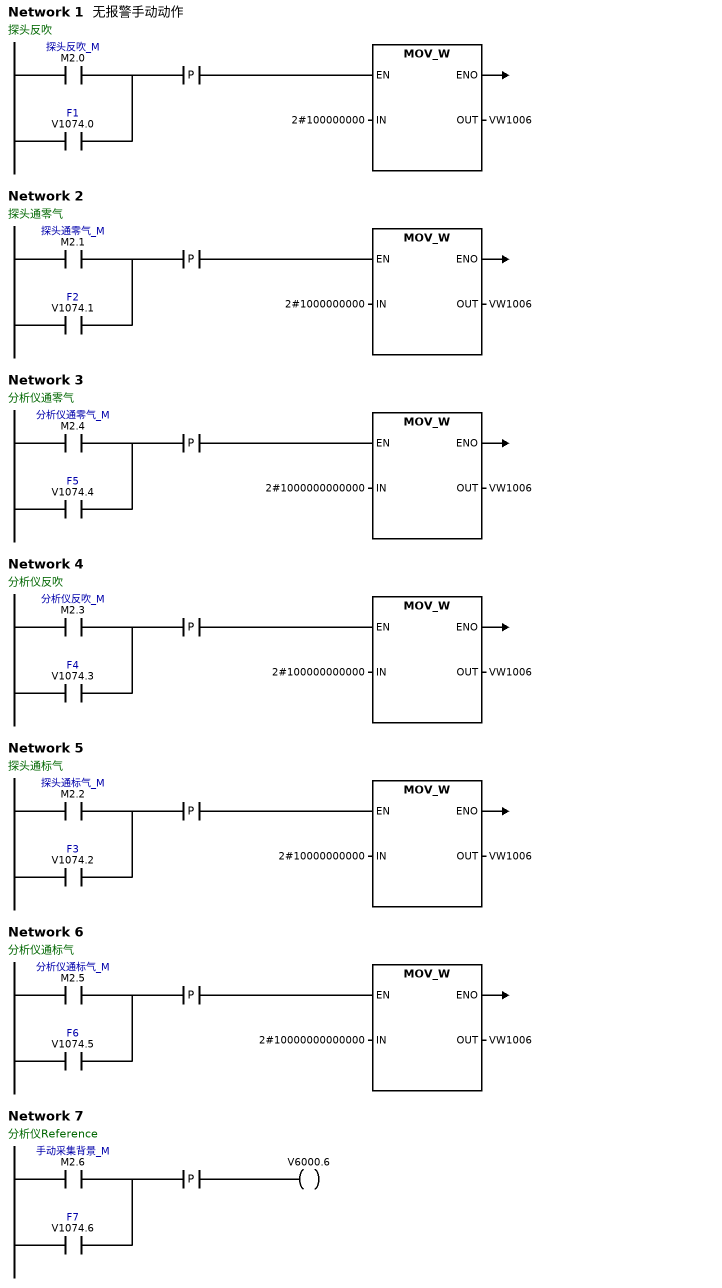
Network 1 // 无报警手动动作
// 探头反吹
LD     探头反吹_M:M2.0
O      F1:V1074.0
EU
MOVW   2#100000000, VW1006
Network 2
// 探头通零气
LD     探头通零气_M:M2.1
O      F2:V1074.1
EU
MOVW   2#1000000000, VW1006
Network 3
// 分析仪通零气
LD     分析仪通零气_M:M2.4
O      F5:V1074.4
EU
MOVW   2#1000000000000, VW1006
Network 4
// 分析仪反吹
LD     分析仪反吹_M:M2.3
O      F4:V1074.3
EU
MOVW   2#100000000000, VW1006
Network 5
// 探头通标气
LD     探头通标气_M:M2.2
O      F3:V1074.2
EU
MOVW   2#10000000000, VW1006
Network 6
// 分析仪通标气
LD     分析仪通标气_M:M2.5
O      F6:V1074.5
EU
MOVW   2#10000000000000, VW1006
Network 7
// 分析仪Reference
LD     手动采集背景_M:M2.6
O      F7:V1074.6
EU
=      V6000.6
END_SUBROUTINE_BLOCK

SUBROUTINE_BLOCK Manual_with_Ana_Alarm:SBR13
TITLE=子程序注释
BEGIN
